{attribute 'GeneratedUsingTerminal: EK1100-0000-0018'}
{attribute addProperty BoxType "EK1100-0000-0018"}
{attribute addProperty Id "Beckhoff_EL3xxx_0030EK1122Beckhoff_EL3xxx_0030EK1122_55DAE3CA2A_0001_EL3174_0030_0016EL3174_DCC7866252A_0002_EL3314_0030_0021EL3314_C9476E1C48A_0003_EL3681_0030_0021EL3681_C165473F32A_0004_EL3201_0030_0022EL3201_F37BFE8521A_0005_EL3202_0030_0022EL3202_27F1223730A_0006_EL3356_0030_0025EL3356_1EAAA6FF28A_0007_EL3692_0030_0021EL3692_E258221652"}
{attribute addProperty CRC "3279650120"}
{attribute addProperty Size "265"}
TYPE Beckhoff_EL3xxx_0030_C37B7D48 EXTENDS EK1100_1FC0878B :
STRUCT
	{attribute addProperty Name "Beckhoff_EL3xxx_0030EK1122"}
	{attribute addProperty PreviousPort "Beckhoff EL3xxx-0030 : B"}
	Beckhoff_EL3xxx_0030EK1122 : Beckhoff_EL3xxx_0030EK1122_55DAE3CA;
	{attribute addProperty Name "A_0001_EL3174_0030_0016"}
	{attribute addProperty PreviousPort "Beckhoff EL3xxx-0030EK1122 : C"}
	A_0001_EL3174_0030_0016 : EL3174_DCC78662;
	{attribute addProperty Name "A_0002_EL3314_0030_0021"}
	{attribute addProperty PreviousPort "A_0001(EL3174-0030-0016) : B"}
	A_0002_EL3314_0030_0021 : EL3314_C9476E1C;
	{attribute addProperty Name "A_0003_EL3681_0030_0021"}
	{attribute addProperty PreviousPort "A_0002(EL3314-0030-0021) : B"}
	A_0003_EL3681_0030_0021 : EL3681_C165473F;
	{attribute addProperty Name "A_0004_EL3201_0030_0022"}
	{attribute addProperty PreviousPort "A_0003(EL3681-0030-0021) : B"}
	A_0004_EL3201_0030_0022 : EL3201_F37BFE85;
	{attribute addProperty Name "A_0005_EL3202_0030_0022"}
	{attribute addProperty PreviousPort "A_0004(EL3201-0030-0022) : B"}
	A_0005_EL3202_0030_0022 : EL3202_27F12237;
	{attribute addProperty Name "A_0006_EL3356_0030_0025"}
	{attribute addProperty PreviousPort "A_0005(EL3202-0030-0022) : B"}
	A_0006_EL3356_0030_0025 : EL3356_1EAAA6FF;
	{attribute addProperty Name "A_0007_EL3692_0030_0021"}
	{attribute addProperty PreviousPort "A_0006(EL3356-0030-0025) : B"}
	A_0007_EL3692_0030_0021 : EL3692_E2582216;
END_STRUCT
END_TYPE

(* stored: Version 1.2.0.0, ProductVersion 3.1.4024.9
   DUT Beckhoff_EL3xxx_0030_C37B7D48: Id {ee1359c0-081a-4fbf-94d9-62643c6f167d} *)
